// TIA Portal V17 export
// export: Created 2024-09-03T21:54:46.9575074Z, ExportSetting WithDefaults, DisplayName Totally Integrated Automation Portal, DisplayVersion V17 Update 7, DisplayName TIA Portal Openness, DisplayVersion V17 Update 7, DisplayName TIA Portal Version Control Interface, DisplayVersion V17, DisplayName SINAMICS Startdrive Advanced, DisplayVersion V17 SP2, DisplayName SINAMICS Startdrive G110M, G120, G120C, G120D, G120P, G115D, DisplayVersion V17 SP2, DisplayName SINAMICS Startdrive G130, G150, S120, S150, SINAMICS MV, S210, DisplayVersion V17 SP2, DisplayName STEP 7 Professional, DisplayVersion V17 Update 7, DisplayName STEP 7 Safety, DisplayVersion V17 Update 6, DisplayName WinCC Advanced / Unified PC, DisplayVersion V17 Update 7
DATA_BLOCK "RobotMain_DB"   // DB17
VERSION : 0.1
// stored: AutoNumber true, DBAccessibleFromOPCUA true, DBAccessibleFromWebserver true, InstanceOfName RobotMain, InstanceOfType FB
"RobotMain"
   // VAR_OUTPUT
   //    RobotInStartingPosition : Bool;
   // END_VAR
   // VAR
   //    R1 { S7_SetPoint := 'True'} : "RobotControl";
   //    R_TRIG_Instance { S7_SetPoint := 'True'} : R_TRIG;
   //    F_TRIG_Instance { S7_SetPoint := 'True'} : F_TRIG;
   // END_VAR
BEGIN
   R1.StartReq := FALSE;
   R1.KeyExt := FALSE;
   R1.JobNrReq := 16#00;
   R1.periReady := FALSE;
   R1.stopMess := TRUE;
   R1.progAct := FALSE;
   R1.onPath := FALSE;
   R1.ext := TRUE;
   R1.internalEstop := FALSE;
   R1.home := TRUE;
   R1.pgNoReq := FALSE;
   R1.robStopped := TRUE;
   R1.jobNrBack := 16#00;
   R1.StartAllowed := FALSE;
   R1.Started := FALSE;
   R1.drivesOn := FALSE;
   R1.confMess := FALSE;
   R1.ExtStart := FALSE;
   R1.moveEnable := TRUE;
   R1.reqHome := FALSE;
   R1.pgNoValid := FALSE;
   R1.reqDoor := FALSE;
   R1.jobNr := 16#00;
   R_TRIG_Instance.CLK := FALSE;
   R_TRIG_Instance.Q := FALSE;
   R_TRIG_Instance.Stat_Bit := FALSE;
   F_TRIG_Instance.CLK := FALSE;
   F_TRIG_Instance.Q := FALSE;
   F_TRIG_Instance.Stat_Bit := FALSE;
END_DATA_BLOCK
